//{attribute 'pack_mode' := '8'}
TYPE ST_ToleranceThresholdPK :
STRUCT
		GoodReadPercentagePAL		:	STRING(6);
		GoodReadPercentageCS		:	STRING(6);
		GoodReadPercentageOUT		:	STRING(6);
END_STRUCT
END_TYPE

(* stored: Version 1.1.0.1
   DUT ST_ToleranceThresholdPK: Id {a4f7e30e-295a-4b82-8431-d9c33017842a} *)
